PROGRAM MAIN
VAR
END_VAR

POU_1();

END_PROGRAM

(* stored: Version 1.1.0.1, ProductVersion 3.1.4024.3
   POU MAIN: Id {3471505b-dea7-49c5-a551-fde9e81c0829}, SpecialFunc None *)
